FUNCTION_BLOCK TokenRingNode (* TokenRing pattern demo: one controller's position in a mutual-exclusion token ring *)
  (* Standard: 61499-2; Description: Copyright (c) 2026 Meisterschulen am Ostbahnhof This program and the accompanying materials are made available under the terms of the Eclipse Public License 2.0 which is available at https://www.eclipse.org/legal/epl-2.0/ SPDX-License-Identifier: EPL-2.0 *)
  (* Version 1.0, 2026-08-31, Franz Höpfinger, Meisterschulen am Ostbahnhof, Mutual Exclusion / TokenRing design pattern (IEC 61499 primer course, Module 6, Valeriy Vyatkin, slide 15), demo node. GIVE/RCV Socket/Plug roles confirmed against Dai/Vyatkin/Christensen/Dubinin, IEEE INDIN 2014, see TokenRingPattern.md *)
  PACKAGE Meins::DesingPatterns::TokenRingPattern;
  (* Documentation:
  One controller's position in a TokenRing / Mutual Exclusion demo ring (IEC 61499 primer course, Module 6, Valeriy Vyatkin, slide 15).
   Has an MTXIN Socket (receives the token from the upstream neighbour, acknowledges with RCV) and an MTXOUT Plug (hands the token to the downstream neighbour with GIVE, reacts to its RCV acknowledgement). On REQUEST it remembers to use the critical section the next time it holds the token; on token arrival it optionally does so (demo: instantaneous, fires ENTERED then EXITED with no real work in between) before passing the token on. SEED bootstraps the ring by injecting the token once, without having received it first - fire it on exactly one node after INIT.
   See TokenRingPattern.md in this folder for the full write-up, including the (unverified) reasoning behind the GIVE/RCV Socket/Plug role split.
  *)
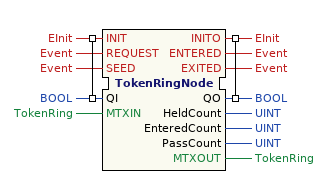
  EVENT_INPUT
    INIT : EInit WITH QI; (* Initialization Request *)
    REQUEST; (* Demo: request the critical section for the next time this node holds the token *)
    SEED; (* Demo: bootstrap the ring by injecting the token here once, on exactly one node, after INIT *)
  END_EVENT
  EVENT_OUTPUT
    INITO : EInit WITH QO; (* Initialization Confirm *)
    ENTERED; (* This node entered its critical section (demo: instantaneous, no real work modelled) *)
    EXITED; (* This node left its critical section and is passing the token on *)
  END_EVENT
  VAR_INPUT
    QI : BOOL; (* Input event qualifier *)
  END_VAR
  VAR_OUTPUT
    QO : BOOL; (* Output event qualifier *)
    HeldCount : UINT; (* Number of times this node received the token (demo counter) *)
    EnteredCount : UINT; (* Number of times this node used the critical section (demo counter) *)
    PassCount : UINT; (* Number of times this node's hand-off was acknowledged (demo counter) *)
  END_VAR
  SOCKETS
    MTXIN : adapter::types::bidirectional::TokenRing::TokenRing; (* Receives the token from the upstream neighbour, acknowledges receipt *)
  END_SOCKETS
  PLUGS
    MTXOUT : adapter::types::bidirectional::TokenRing::TokenRing; (* Hands the token to the downstream neighbour, waits for its acknowledgement *)
  END_PLUGS
  VAR
    Want : BOOL; (* Critical section requested for the next token hold *)
  END_VAR
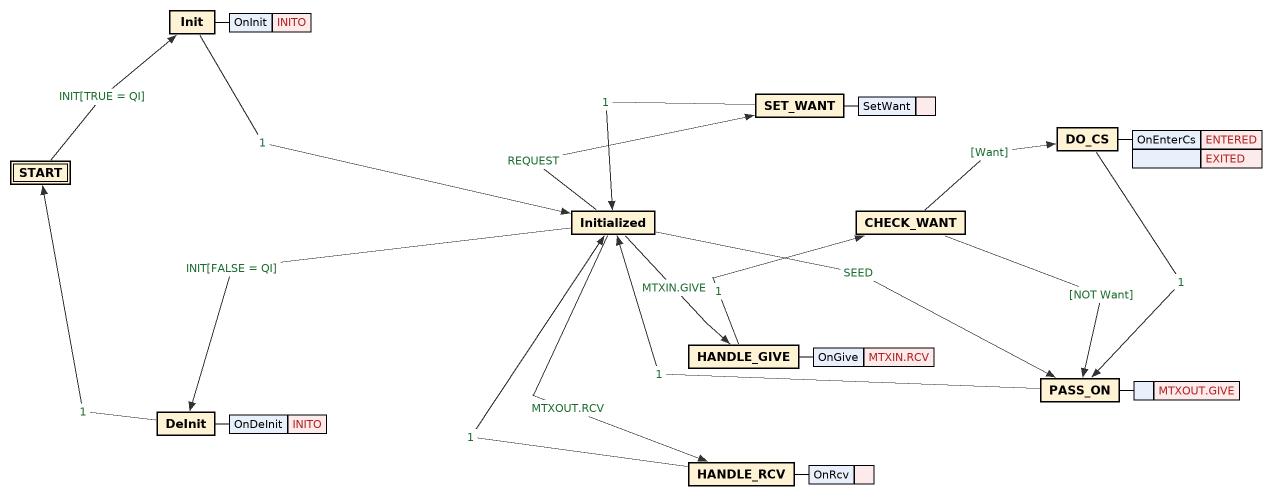
  EC_STATES
    START; (* Uninitialized *)
    Init : OnInit -> INITO; (* Initialization *)
    Initialized; (* Idle, waiting for the token or a local request *)
    DeInit : OnDeInit -> INITO; (* De-initialization *)
    SET_WANT : SetWant; (* Remember that this node wants the critical section next time it holds the token *)
    HANDLE_GIVE : OnGive -> MTXIN.RCV; (* Token arrived: count it, acknowledge receipt *)
    CHECK_WANT; (* Decide whether to use the critical section before passing the token on *)
    DO_CS : OnEnterCs -> ENTERED, -> EXITED; (* Use the critical section (demo: instantaneous) *)
    PASS_ON : -> MTXOUT.GIVE; (* Hand the token to the downstream neighbour *)
    HANDLE_RCV : OnRcv; (* Downstream neighbour acknowledged receipt *)
  END_STATES
  EC_TRANSITIONS
    START TO Init := INIT[TRUE = QI];
    Init TO Initialized := 1;
    Initialized TO DeInit := INIT[FALSE = QI];
    DeInit TO START := 1;
    Initialized TO SET_WANT := REQUEST;
    SET_WANT TO Initialized := 1;
    Initialized TO HANDLE_GIVE := MTXIN.GIVE;
    HANDLE_GIVE TO CHECK_WANT := 1;
    CHECK_WANT TO DO_CS := [Want];
    CHECK_WANT TO PASS_ON := [NOT Want];
    Initialized TO PASS_ON := SEED;
    DO_CS TO PASS_ON := 1;
    PASS_ON TO Initialized := 1;
    Initialized TO HANDLE_RCV := MTXOUT.RCV;
    HANDLE_RCV TO Initialized := 1;
  END_TRANSITIONS
  ALGORITHM OnInit IN ST: (* Reset demo counters/flags *)
HeldCount := 0;
EnteredCount := 0;
PassCount := 0;
Want := FALSE;
QO := QI;
  END_ALGORITHM
  ALGORITHM OnDeInit IN ST: (* De-initialize *)
QO := FALSE;
  END_ALGORITHM
  ALGORITHM SetWant IN ST: (* Remember to use the critical section next time the token arrives *)
Want := TRUE;
  END_ALGORITHM
  ALGORITHM OnGive IN ST: (* Count a received token *)
HeldCount := HeldCount + 1;
  END_ALGORITHM
  ALGORITHM OnEnterCs IN ST: (* Count and clear the pending request *)
EnteredCount := EnteredCount + 1;
Want := FALSE;
  END_ALGORITHM
  ALGORITHM OnRcv IN ST: (* Count an acknowledged hand-off *)
PassCount := PassCount + 1;
  END_ALGORITHM
END_FUNCTION_BLOCK
